// SIMATIC STEP 7 (V5.x) project PUT_GET
// program: S7 Program(1)

SYMBOL_TABLE
"RCV_DATA"	DB 10	DB 10
"SND_DATA"	DB 11	DB 11
"FB_COM"	FB 330	FB 330
"COM_INIT"	FC 100	FC 100
"COM_RES"	FC 101	FC 101
END_SYMBOL_TABLE

FUNCTION_BLOCK "FB_COM"	// FB 330
VERSION : 0.1
VAR_INPUT
  INIT_COM : BOOL ;
END_VAR
VAR
  PLC1_COM : STRUCT
   GET_REQ : BOOL ;
   GET_BUSY : BOOL ;
   GET_NDR : BOOL ;
   GET_ERROR : BOOL ;
   GET_START : BOOL ;	//Pos flank
   PUT_REQ : BOOL ;
   PUT_BUSY : BOOL ;
   PUT_DONE : BOOL ;
   PUT_ERROR : BOOL ;
   PUT_START : BOOL ;
   ID : WORD ;
   GET_STATUS : WORD ;
   GET_STAT_SAVE : WORD ;
   PUT_STATUS : WORD ;
   PUT_STAT_SAVE : WORD ;
  END_STRUCT ;
  Statistic : STRUCT
   GET_NDR : INT ;
   GET_ERROR : INT ;
   PUT_DONE : INT ;
   PUT_ERROR : INT ;
  END_STRUCT ;
  PLC_GET : FB 14;
  PLC_PUT : FB 15;
  STAT0 : BOOL ;
END_VAR
BEGIN
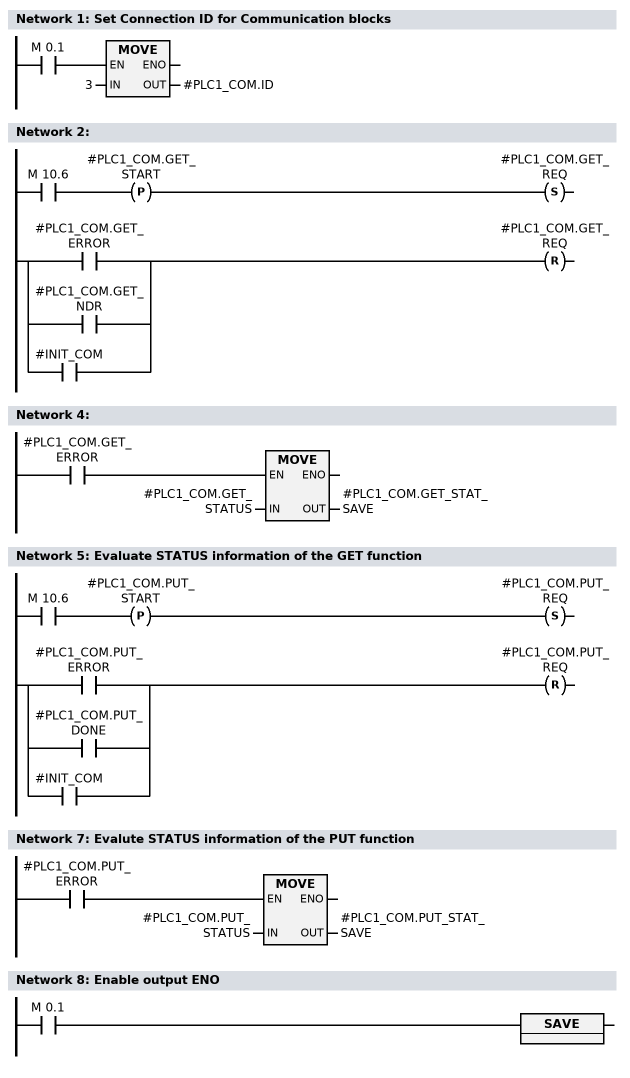
NETWORK
TITLE = Set Connection ID for Communication blocks
      A     M 0.1;
      JNB   _004;
      L     3;
      T     #PLC1_COM.ID;
_004: NOP   0;
NETWORK
TITLE =
//Start GET function with the rising edge of the clock marker if GET function is 
//not BUSY.
      A     M 10.6;
      FP    #PLC1_COM.GET_START;
      S     #PLC1_COM.GET_REQ;
      A(;
      O     #PLC1_COM.GET_ERROR;
      O     #PLC1_COM.GET_NDR;
      O     #INIT_COM;
      );
      R     #PLC1_COM.GET_REQ;
      NOP   0;
NETWORK
TITLE = Invoke GET function
      A     #PLC1_COM.GET_REQ;
      =     L 0.0;
      BLD   103;
      A     M 0.1;
      JNB   _005;
      BLD   14;
      =     L 7.0;
      L     DINO;
      T     LW 5;
      CDB;
      OPN   DI [LW 5];
      TAR2  LD 1;
      A     L 0.0;
      =     DIX [AR2,P#22.0];
      L     DBW [AR2,P#4.0];
      T     DIW [AR2,P#24.0];
      L     W#16#1002;
      T     DIW [AR2,P#30.0];
      L     26;
      T     DIW [AR2,P#32.0];
      L     11;
      T     DIW [AR2,P#34.0];
      L     P#DBX 0.0;
      T     DID [AR2,P#36.0];
      L     W#16#1002;
      T     DIW [AR2,P#40.0];
      L     26;
      T     DIW [AR2,P#42.0];
      L     10;
      T     DIW [AR2,P#44.0];
      L     P#DBX 0.0;
      T     DID [AR2,P#46.0];
      +AR2  P#22.0;
      UC    FB 14;
      LAR2  LD 1;
      A     DIX [AR2,P#26.0];
      =     DBX [AR2,P#2.2];
      A     DIX [AR2,P#26.1];
      =     DBX [AR2,P#2.3];
      L     DIW [AR2,P#28.0];
      T     DBW [AR2,P#6.0];
      CDB;
      BLD   15;
_005: NOP   0;
NETWORK
TITLE =
//If ERROR occured then save STATUS!
//
      A     #PLC1_COM.GET_ERROR;
      JNB   _006;
      L     #PLC1_COM.GET_STATUS;
      T     #PLC1_COM.GET_STAT_SAVE;
_006: NOP   0;
NETWORK
TITLE = Evaluate STATUS information of the GET function
//Start PUT function with the rising edge of the clock marker if PUT function is 
//not BUSY.
//
      A     M 10.6;
      FP    #PLC1_COM.PUT_START;
      S     #PLC1_COM.PUT_REQ;
      A(;
      O     #PLC1_COM.PUT_ERROR;
      O     #PLC1_COM.PUT_DONE;
      O     #INIT_COM;
      );
      R     #PLC1_COM.PUT_REQ;
      NOP   0;
NETWORK
TITLE = Invoke PUT function
      A     #PLC1_COM.PUT_REQ;
      =     L 0.0;
      BLD   103;
      A     M 0.1;
      JNB   _007;
      BLD   14;
      =     L 7.0;
      L     DINO;
      T     LW 5;
      CDB;
      OPN   DI [LW 5];
      TAR2  LD 1;
      A     L 0.0;
      =     DIX [AR2,P#466.0];
      L     DBW [AR2,P#4.0];
      T     DIW [AR2,P#468.0];
      L     W#16#1002;
      T     DIW [AR2,P#474.0];
      L     26;
      T     DIW [AR2,P#476.0];
      L     10;
      T     DIW [AR2,P#478.0];
      L     P#DBX 0.0;
      T     DID [AR2,P#480.0];
      L     W#16#1002;
      T     DIW [AR2,P#484.0];
      L     26;
      T     DIW [AR2,P#486.0];
      L     11;
      T     DIW [AR2,P#488.0];
      L     P#DBX 0.0;
      T     DID [AR2,P#490.0];
      +AR2  P#466.0;
      UC    FB 15;
      LAR2  LD 1;
      A     DIX [AR2,P#470.0];
      =     DBX [AR2,P#2.7];
      A     DIX [AR2,P#470.1];
      =     DBX [AR2,P#3.0];
      L     DIW [AR2,P#472.0];
      T     DBW [AR2,P#10.0];
      CDB;
      BLD   15;
_007: NOP   0;
NETWORK
TITLE = Evalute STATUS information of the PUT function
//If ERROR occured then save STATUS,
//if DONE signals completion then reset BUSY for the next cycle!
      A     #PLC1_COM.PUT_ERROR;
      JNB   _008;
      L     #PLC1_COM.PUT_STATUS;
      T     #PLC1_COM.PUT_STAT_SAVE;
_008: NOP   0;
NETWORK
TITLE = Enable output ENO
      A     M 0.1;
      SAVE;
END_FUNCTION_BLOCK

FUNCTION "COM_INIT" : VOID	// FC 100
//For OB100
VERSION : 0.1
BEGIN
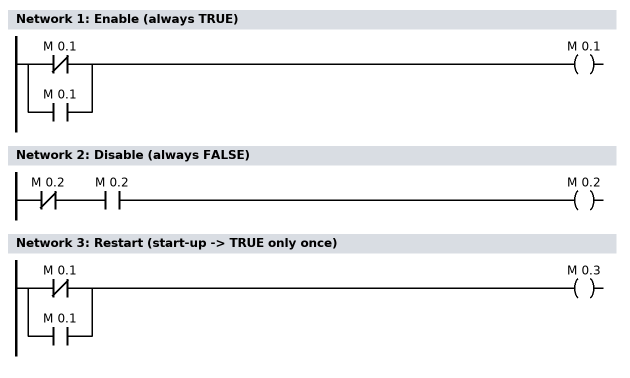
NETWORK
TITLE = Enable (always TRUE)
      ON    M 0.1;
      O     M 0.1;
      =     M 0.1;
NETWORK
TITLE = Disable (always FALSE)
      AN    M 0.2;
      A     M 0.2;
      =     M 0.2;
NETWORK
TITLE = Restart (start-up -> TRUE only once)
      ON    M 0.1;
      O     M 0.1;
      =     M 0.3;
END_FUNCTION

FUNCTION "COM_RES" : VOID	// FC 101
TITLE = Reset initial communication start
VERSION : 0.1
BEGIN
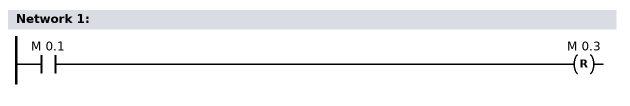
NETWORK
TITLE =
      A     M 0.1;
      R     M 0.3;
END_FUNCTION

DATA_BLOCK "RCV_DATA"	// DB 10
VERSION : 0.1
  STRUCT
   N11_1_2_QAUTO : BOOL ;	//Рабочий насос N11 в автомате
   N11_1_2_QPAZ : BOOL ;
   N11_1_2_QFAULT : BOOL ;	//Авария насосов N11
   N11_1_2_ON_ACK : BOOL ;	//Подтверждение включения рабочего насоса N11
   N11_1_2_OFF_ACK : BOOL ;	//Подтверждение отключения рабочего насоса N11
   test : BOOL ;
   res_bit4 : BOOL ;
   res_bit5 : BOOL ;
   res_bit6 : BOOL ;
   res_bit7 : BOOL ;
   res_bit8 : BOOL ;
   res_bit9 : BOOL ;
   res_bit10 : BOOL ;
   res_bit11 : BOOL ;
   res_bit12 : BOOL ;
   res_bit13 : BOOL ;
   res_word : INT ;
   res_word1 : INT ;
   res_word2 : INT ;
   res_word3 : INT ;
   res_dword : REAL ;
   res_dword1 : REAL ;
   res_dword2 : REAL ;
   res_dword3 : REAL ;
  END_STRUCT ;	
BEGIN
END_DATA_BLOCK

DATA_BLOCK "SND_DATA"	// DB 11
VERSION : 0.1
  STRUCT
   N11_1_2_ON : BOOL ;	//Команда на включение насоса 11N-1 11N-2
   N11_1_2_OFF : BOOL ;	//Команда на отключение насоса 11N-1 11N-2
   res_bit13 : BOOL ;
   res_bit12 : BOOL ;
   res_bit : BOOL ;
   res_bit1 : BOOL ;
   res_bit2 : BOOL ;
   res_bit3 : BOOL ;
   res_bit4 : BOOL ;
   res_bit5 : BOOL ;
   res_bit6 : BOOL ;
   res_bit7 : BOOL ;
   res_bit8 : BOOL ;
   res_bit9 : BOOL ;
   res_bit10 : BOOL ;
   res_bit11 : BOOL ;
   res_word : INT ;
   res_word1 : INT ;
   res_word2 : INT ;
   res_word3 : INT ;
   res_dword : REAL ;
   res_dword1 : REAL ;
   res_dword2 : REAL ;
   res_dword3 : REAL ;
  END_STRUCT ;	
BEGIN
END_DATA_BLOCK

ORGANIZATION_BLOCK OB 1
TITLE = "Main Program Sweep (Cycle)"
VERSION : 0.1
VAR_TEMP
  OB1_EV_CLASS : BYTE ;	//Bits 0-3 = 1 (Coming event), Bits 4-7 = 1 (Event class 1)
  OB1_SCAN_1 : BYTE ;	//1 (Cold restart scan 1 of OB 1), 3 (Scan 2-n of OB 1)
  OB1_PRIORITY : BYTE ;	//Priority of OB Execution
  OB1_OB_NUMBR : BYTE ;	//1 (Organization block 1, OB1)
  OB1_RESERVED_1 : BYTE ;	//Reserved for system
  OB1_RESERVED_2 : BYTE ;	//Reserved for system
  OB1_PREV_CYCLE : INT ;	//Cycle time of previous OB1 scan (milliseconds)
  OB1_MIN_CYCLE : INT ;	//Minimum cycle time of OB1 (milliseconds)
  OB1_MAX_CYCLE : INT ;	//Maximum cycle time of OB1 (milliseconds)
  OB1_DATE_TIME : DATE_AND_TIME ;	//Date and time OB1 started
END_VAR
BEGIN
// (block stored without names or comments; labels and parameter names are numbered)
END_ORGANIZATION_BLOCK
